LIN {X 5.578,Y -23.911,Z -42.731,A 0.015,B -0.000,C 180.000} C_DIS
LIN {X 5.597,Y -23.749,Z -43.353,A 0.015,B 0.000,C 180.000} C_DIS
LIN {X 5.625,Y -23.303,Z -43.816,A 0.015,B 0.000,C -180.000} C_DIS
LIN {X 5.610,Y -22.688,Z -44.000,A 0.015,B 0.000,C -180.000} C_DIS
LIN {X 1.585,Y -17.451,Z -44.244,A 0.015,B 0.000,C 180.000} C_DIS
LIN {X -4.825,Y -19.040,Z -44.488,A 0.015,B -0.000,C 180.000} C_DIS
LIN {X -5.938,Y -25.550,Z -44.732,A 0.015,B 0.000,C -180.000} C_DIS
LIN {X -0.420,Y -29.178,Z -44.976,A 0.015,B 0.000,C 180.000} C_DIS
LIN {X 5.116,Y -25.576,Z -45.220,A 0.015,B 0.000,C -180.000} C_DIS
LIN {X 4.034,Y -19.061,Z -45.464,A 0.015,B 0.000,C 180.000} C_DIS
LIN {X -2.368,Y -17.441,Z -45.708,A 0.015,B 0.000,C 180.000} C_DIS
LIN {X -6.418,Y -22.658,Z -45.952,A 0.015,B 0.000,C 180.000} C_DIS
LIN {X -3.261,Y -28.459,Z -46.196,A 0.015,B 0.000,C -180.000} C_DIS
LIN {X 3.319,Y -27.891,Z -46.440,A 0.015,B -0.000,C 180.000} C_DIS
LIN {X 5.435,Y -21.635,Z -46.685,A 0.015,B 0.000,C 180.000} C_DIS
LIN {X 0.551,Y -17.189,Z -46.929,A 0.015,B 0.000,C -180.000} C_DIS
LIN {X -5.479,Y -19.882,Z -47.173,A 0.015,B 0.000,C 180.000} C_DIS
LIN {X -5.428,Y -26.486,Z -47.417,A 0.015,B 0.000,C 180.000} C_DIS
LIN {X 0.643,Y -29.086,Z -47.661,A 0.015,B -0.000,C -180.000} C_DIS
LIN {X 5.458,Y -24.566,Z -47.905,A 0.015,B 0.000,C 180.000} C_DIS
LIN {X 3.245,Y -18.343,Z -48.149,A 0.015,B 0.000,C 180.000} C_DIS
LIN {X -3.342,Y -17.876,Z -48.393,A 0.015,B 0.000,C 180.000} C_DIS
LIN {X -6.410,Y -23.725,Z -48.637,A 0.015,B 0.000,C 180.000} C_DIS
LIN {X -2.281,Y -28.879,Z -48.881,A 0.015,B 0.000,C 180.000} C_DIS
LIN {X 4.096,Y -27.161,Z -49.125,A 0.015,B 0.000,C -180.000} C_DIS
LIN {X 5.078,Y -20.630,Z -49.369,A 0.015,B 0.000,C 180.000} C_DIS
LIN {X -0.513,Y -17.114,Z -49.613,A 0.015,B 0.000,C 180.000} C_DIS
LIN {X -5.974,Y -20.827,Z -49.857,A 0.015,B -0.000,C 180.000} C_DIS
LIN {X -4.761,Y -27.319,Z -50.101,A 0.015,B 0.000,C -180.000} C_DIS
LIN {X 1.673,Y -28.809,Z -50.345,A 0.015,B 0.000,C -180.000} C_DIS
LIN {X 5.616,Y -23.511,Z -50.589,A 0.015,B 0.000,C -180.000} C_DIS
LIN {X 2.342,Y -17.775,Z -50.833,A 0.015,B 0.000,C -180.000} C_DIS
LIN {X -4.225,Y -18.476,Z -51.077,A 0.015,B 0.000,C 180.000} C_DIS
LIN {X -6.214,Y -24.774,Z -51.321,A 0.015,B 0.000,C 180.000} C_DIS
LIN {X -1.241,Y -29.120,Z -51.565,A 0.015,B 0.000,C 180.000} C_DIS
LIN {X 4.733,Y -26.306,Z -51.810,A 0.015,B 0.000,C -180.000} C_DIS
LIN {X 4.549,Y -19.704,Z -52.054,A 0.015,B -0.000,C 180.000} C_DIS
LIN {X -1.573,Y -17.227,Z -52.298,A 0.015,B 0.000,C 180.000} C_DIS
LIN {X -6.296,Y -21.844,Z -52.542,A 0.015,B 0.000,C -180.000} C_DIS
LIN {X -3.958,Y -28.021,Z -52.786,A 0.015,B 0.000,C 180.000} C_DIS
LIN {X 2.638,Y -28.354,Z -53.030,A 0.015,B 0.000,C 180.000} C_DIS
LIN {X 5.586,Y -22.445,Z -53.274,A 0.015,B 0.000,C 180.000} C_DIS
LIN {X 1.354,Y -17.375,Z -53.518,A 0.015,B -0.000,C 180.000} C_DIS
LIN {X -4.987,Y -19.222,Z -53.762,A 0.015,B 0.000,C 180.000} C_DIS
LIN {X -5.836,Y -25.771,Z -54.006,A 0.015,B 0.000,C 180.000} C_DIS
LIN {X -0.176,Y -29.174,Z -54.250,A 0.015,B 0.000,C -180.000} C_DIS
LIN {X 5.210,Y -25.351,Z -54.494,A 0.015,B -0.000,C 180.000} C_DIS
LIN {X 3.865,Y -18.885,Z -54.738,A 0.015,B -0.000,C -180.000} C_DIS
LIN {X -2.597,Y -17.525,Z -54.982,A 0.015,B 0.000,C 180.000} C_DIS
LIN {X -6.433,Y -22.902,Z -55.226,A 0.015,B 0.000,C -180.000} C_DIS
LIN {X -3.044,Y -28.570,Z -55.470,A 0.015,B 0.000,C -180.000} C_DIS
LIN {X 3.508,Y -27.737,Z -55.714,A 0.015,B 0.000,C -180.000} C_DIS
LIN {X 5.369,Y -21.401,Z -55.958,A 0.015,B 0.000,C 180.000} C_DIS
LIN {X 0.310,Y -17.156,Z -56.202,A 0.015,B -0.000,C 180.000} C_DIS
LIN {X -5.607,Y -20.090,Z -56.446,A 0.015,B 0.000,C 180.000} C_DIS
LIN {X -5.289,Y -26.687,Z -56.690,A 0.015,B 0.000,C -180.000} C_DIS
LIN {X 0.882,Y -29.039,Z -56.935,A 0.015,B 0.000,C 180.000} C_DIS
LIN {X 5.510,Y -24.328,Z -57.179,A 0.015,B 0.000,C 180.000} C_DIS
LIN {X 3.048,Y -18.200,Z -57.423,A 0.015,B -0.000,C 180.000} C_DIS
LIN {X -3.553,Y -17.999,Z -57.667,A 0.015,B 0.000,C 180.000} C_DIS
LIN {X -6.382,Y -23.967,Z -57.911,A 0.015,B 0.000,C -180.000} C_DIS
LIN {X -2.047,Y -28.950,Z -58.155,A 0.015,B 0.000,C 180.000} C_DIS
LIN {X 4.255,Y -26.976,Z -58.399,A 0.015,B 0.000,C 180.000} C_DIS
LIN {X 4.972,Y -20.411,Z -58.643,A 0.015,B 0.000,C 180.000} C_DIS
LIN {X -0.756,Y -17.123,Z -58.887,A 0.015,B 0.000,C 180.000} C_DIS
LIN {X -6.064,Y -21.054,Z -59.131,A 0.015,B 0.000,C 180.000} C_DIS
LIN {X -4.589,Y -27.492,Z -59.375,A 0.015,B 0.000,C -180.000} C_DIS
LIN {X 1.900,Y -28.720,Z -59.619,A 0.015,B 0.000,C 180.000} C_DIS
LIN {X 5.626,Y -23.267,Z -59.863,A 0.015,B 0.000,C 180.000} C_DIS
LIN {X 2.123,Y -17.669,Z -60.107,A 0.015,B 0.000,C -180.000} C_DIS
LIN {X -4.410,Y -18.634,Z -60.351,A 0.015,B 0.000,C 180.000} C_DIS
LIN {X -6.143,Y -25.007,Z -60.595,A 0.015,B 0.000,C -180.000} C_DIS
LIN {X -0.999,Y -29.149,Z -60.839,A 0.015,B 0.000,C 180.000} C_DIS
LIN {X 4.857,Y -26.095,Z -61.083,A 0.015,B 0.000,C -180.000} C_DIS
LIN {X 4.406,Y -19.506,Z -61.327,A 0.015,B 0.000,C -180.000} C_DIS
LIN {X -1.812,Y -17.279,Z -61.571,A 0.015,B 0.000,C 180.000} C_DIS
LIN {X -6.344,Y -22.083,Z -61.815,A 0.015,B -0.000,C -180.000} C_DIS
LIN {X -3.758,Y -28.161,Z -62.060,A 0.015,B -0.000,C 180.000} C_DIS
LIN {X 2.846,Y -28.227,Z -62.304,A 0.015,B 0.000,C 180.000} C_DIS
LIN {X 5.553,Y -22.203,Z -62.548,A 0.015,B -0.000,C -180.000} C_DIS
LIN {X 1.119,Y -17.309,Z -62.792,A 0.015,B 0.000,C 180.000} C_DIS
LIN {X -5.142,Y -19.410,Z -63.036,A 0.015,B 0.000,C -180.000} C_DIS
LIN {X -5.726,Y -25.989,Z -63.280,A 0.015,B -0.000,C 180.000} C_DIS
LIN {X 0.067,Y -29.160,Z -63.524,A 0.015,B -0.000,C -180.000} C_DIS
LIN {X 5.294,Y -25.122,Z -63.768,A 0.015,B 0.000,C -180.000} C_DIS
LIN {X 3.690,Y -18.716,Z -64.012,A 0.015,B 0.000,C -180.000} C_DIS
LIN {X -2.823,Y -17.619,Z -64.256,A 0.015,B 0.000,C 180.000} C_DIS
LIN {X -6.438,Y -23.146,Z -64.500,A 0.015,B -0.000,C -180.000} C_DIS
CIRC {X -0.832,Y -28.751,Z -64.500,A 0.015,B 0.000,C -180.000},{X 4.774,Y -23.145,Z -64.500,A 0.015,B 0.000,C 180.000} C_DIS
LIN {X 4.774,Y -20.361,Z -64.500,A 0.015,B 0.000,C -180.000} C_DIS
CIRC {X 3.668,Y -18.804,Z -64.500,A 0.015,B 0.000,C -180.000},{X 1.834,Y -19.336,Z -64.500,A 0.015,B -0.000,C -180.000} C_DIS
LIN {X -0.747,Y -22.588,Z -64.500,A 0.015,B -0.000,C 180.000} C_DIS
CIRC {X -0.977,Y -24.658,Z -64.500,A 0.015,B 0.000,C 180.000},{X 0.787,Y -25.765,Z -64.500,A 0.015,B -0.000,C 180.000} C_DIS
LIN {X 2.660,Y -25.765,Z -64.500,A 0.015,B 0.000,C -180.000} C_DIS
CIRC {X 4.155,Y -25.146,Z -64.500,A 0.015,B -0.000,C 180.000},{X 4.774,Y -23.651,Z -64.500,A 0.015,B 0.000,C -180.000} C_DIS
LIN {X 4.774,Y -23.145,Z -64.500,A 0.015,B -0.000,C 180.000} C_DIS
LIN {X 3.563,Y -23.413,Z -64.500,A 0.015,B 0.000,C 180.000} C_DIS
LIN {X 4.057,Y -24.474,Z -64.500,A 0.015,B 0.000,C 180.000} C_DIS
LIN {X 4.252,Y -24.715,Z -64.500,A 0.015,B 0.000,C -180.000} C_DIS
LIN {X 8.679,Y -28.027,Z -64.500,A 0.015,B -0.000,C 180.000} C_DIS
LIN {X 9.366,Y -28.668,Z -64.500,A 0.015,B 0.000,C -180.000} C_DIS
LIN {X 9.675,Y -28.604,Z -64.500,A 0.015,B 0.000,C -180.000} C_DIS
LIN {X 10.021,Y -27.803,Z -64.500,A 0.015,B 0.000,C -180.000} C_DIS
LIN {X 10.218,Y -26.938,Z -64.500,A 0.015,B -0.000,C 180.000} C_DIS
LIN {X 10.275,Y -25.867,Z -64.500,A 0.015,B 0.000,C -180.000} C_DIS
LIN {X 10.274,Y 7.389,Z -64.500,A 0.015,B -0.000,C 180.000} C_DIS
LIN {X 6.193,Y -2.899,Z -64.500,A 0.015,B 0.000,C -180.000} C_DIS
LIN {X 5.976,Y -3.347,Z -64.500,A 0.015,B 0.000,C 180.000} C_DIS
LIN {X 1.986,Y -10.239,Z -64.500,A 0.015,B -0.000,C 180.000} C_DIS
LIN {X 1.708,Y -10.647,Z -64.500,A 0.015,B -0.000,C 180.000} C_DIS
LIN {X -5.904,Y -20.237,Z -64.500,A 0.015,B 0.000,C -180.000} C_DIS
LIN {X -6.318,Y -20.673,Z -64.500,A 0.015,B -0.000,C -180.000} C_DIS
LIN {X -7.322,Y -21.557,Z -64.500,A 0.015,B -0.000,C 180.000} C_DIS
LIN {X -7.657,Y -21.816,Z -64.500,A 0.015,B -0.000,C 180.000} C_DIS
LIN {X -17.247,Y -28.331,Z -64.500,A 0.015,B 0.000,C 180.000} C_DIS
LIN {X -17.736,Y -28.607,Z -64.500,A 0.015,B 0.000,C -180.000} C_DIS
LIN {X -19.187,Y -29.273,Z -64.500,A 0.015,B 0.000,C -180.000} C_DIS
LIN {X -19.614,Y -29.435,Z -64.500,A 0.015,B -0.000,C 180.000} C_DIS
LIN {X -25.630,Y -31.266,Z -64.500,A 0.015,B 0.000,C 180.000} C_DIS
LIN {X 5.412,Y -31.266,Z -64.500,A 0.015,B 0.000,C 180.000} C_DIS
LIN {X 6.622,Y -31.073,Z -64.500,A 0.015,B 0.000,C 180.000} C_DIS
$VEL.CP = 1.00000
LIN {X 6.622,Y -31.073,Z 11.769,A 0.015,B 0.000,C -180.000} C_DIS
$VEL.CP = 1.00000
LIN {X -399.068,Y -22.363,Z 11.769,A 0.015,B 0.000,C -180.000} C_DIS
$VEL.CP = 0.10000
LIN {X -399.086,Y -22.525,Z 11.147,A 0.015,B 0.000,C -180.000} C_DIS
LIN {X -399.115,Y -22.971,Z 10.684,A 0.015,B -0.000,C 180.000} C_DIS
LIN {X -399.099,Y -23.586,Z 10.500,A 0.015,B -0.000,C -180.000} C_DIS
LIN {X -395.075,Y -28.823,Z 10.256,A 0.015,B 0.000,C 180.000} C_DIS
LIN {X -388.665,Y -27.234,Z 10.012,A 0.015,B -0.000,C 180.000} C_DIS
LIN {X -387.551,Y -20.725,Z 9.768,A 0.015,B 0.000,C 180.000} C_DIS
LIN {X -393.069,Y -17.096,Z 9.524,A 0.015,B 0.000,C 180.000} C_DIS
LIN {X -398.605,Y -20.698,Z 9.280,A 0.015,B -0.000,C 180.000} C_DIS
LIN {X -397.524,Y -27.213,Z 9.036,A 0.015,B -0.000,C -180.000} C_DIS
LIN {X -391.121,Y -28.833,Z 8.792,A 0.015,B 0.000,C -180.000} C_DIS
LIN {X -387.071,Y -23.616,Z 8.548,A 0.015,B -0.000,C -180.000} C_DIS
LIN {X -390.228,Y -17.815,Z 8.304,A 0.015,B 0.000,C -180.000} C_DIS
LIN {X -396.808,Y -18.383,Z 8.060,A 0.015,B 0.000,C 180.000} C_DIS
LIN {X -398.925,Y -24.639,Z 7.815,A 0.015,B 0.000,C -180.000} C_DIS
LIN {X -394.041,Y -29.085,Z 7.571,A 0.015,B -0.000,C -180.000} C_DIS
LIN {X -388.011,Y -26.392,Z 7.327,A 0.015,B -0.000,C -180.000} C_DIS
LIN {X -388.061,Y -19.788,Z 7.083,A 0.015,B -0.000,C -180.000} C_DIS
LIN {X -394.132,Y -17.188,Z 6.839,A 0.015,B 0.000,C 180.000} C_DIS
LIN {X -398.947,Y -21.708,Z 6.595,A 0.015,B 0.000,C 180.000} C_DIS
LIN {X -396.735,Y -27.931,Z 6.351,A 0.015,B 0.000,C 180.000} C_DIS
LIN {X -390.147,Y -28.398,Z 6.107,A 0.015,B -0.000,C 180.000} C_DIS
LIN {X -387.080,Y -22.549,Z 5.863,A 0.015,B 0.000,C 180.000} C_DIS
LIN {X -391.209,Y -17.395,Z 5.619,A 0.015,B -0.000,C -180.000} C_DIS
LIN {X -397.586,Y -19.113,Z 5.375,A 0.015,B -0.000,C -180.000} C_DIS
LIN {X -398.567,Y -25.644,Z 5.131,A 0.015,B -0.000,C -180.000} C_DIS
LIN {X -392.977,Y -29.160,Z 4.887,A 0.015,B 0.000,C -180.000} C_DIS
LIN {X -387.515,Y -25.447,Z 4.643,A 0.015,B 0.000,C 180.000} C_DIS
LIN {X -388.728,Y -18.955,Z 4.399,A 0.015,B 0.000,C -180.000} C_DIS
LIN {X -395.162,Y -17.465,Z 4.155,A 0.015,B -0.000,C -180.000} C_DIS
LIN {X -399.106,Y -22.763,Z 3.911,A 0.015,B -0.000,C 180.000} C_DIS
LIN {X -395.832,Y -28.499,Z 3.667,A 0.015,B 0.000,C 180.000} C_DIS
LIN {X -389.265,Y -27.798,Z 3.423,A 0.015,B 0.000,C -180.000} C_DIS
LIN {X -387.275,Y -21.501,Z 3.179,A 0.015,B -0.000,C 180.000} C_DIS
LIN {X -392.248,Y -17.154,Z 2.935,A 0.015,B -0.000,C -180.000} C_DIS
LIN {X -398.223,Y -19.968,Z 2.690,A 0.015,B -0.000,C -180.000} C_DIS
LIN {X -398.039,Y -26.570,Z 2.446,A 0.015,B 0.000,C -180.000} C_DIS
LIN {X -391.916,Y -29.047,Z 2.202,A 0.015,B 0.000,C -180.000} C_DIS
LIN {X -387.194,Y -24.430,Z 1.958,A 0.015,B 0.000,C -180.000} C_DIS
LIN {X -389.531,Y -18.253,Z 1.714,A 0.015,B 0.000,C -180.000} C_DIS
LIN {X -396.127,Y -17.920,Z 1.470,A 0.015,B 0.000,C -180.000} C_DIS
LIN {X -399.076,Y -23.829,Z 1.226,A 0.015,B -0.000,C 180.000} C_DIS
LIN {X -394.843,Y -28.899,Z 0.982,A 0.015,B 0.000,C 180.000} C_DIS
LIN {X -388.502,Y -27.052,Z 0.738,A 0.015,B 0.000,C -180.000} C_DIS
LIN {X -387.653,Y -20.503,Z 0.494,A 0.015,B -0.000,C 180.000} C_DIS
LIN {X -393.313,Y -17.100,Z 0.250,A 0.015,B 0.000,C -180.000} C_DIS
LIN {X -398.699,Y -20.923,Z 0.006,A 0.015,B 0.000,C 180.000} C_DIS
LIN {X -397.355,Y -27.389,Z -0.238,A 0.015,B -0.000,C -180.000} C_DIS
LIN {X -390.892,Y -28.749,Z -0.482,A 0.015,B 0.000,C -180.000} C_DIS
LIN {X -387.057,Y -23.372,Z -0.726,A 0.015,B 0.000,C 180.000} C_DIS
LIN {X -390.445,Y -17.704,Z -0.970,A 0.015,B -0.000,C 180.000} C_DIS
LIN {X -396.997,Y -18.537,Z -1.214,A 0.015,B 0.000,C 180.000} C_DIS
LIN {X -398.859,Y -24.874,Z -1.458,A 0.015,B 0.000,C -180.000} C_DIS
LIN {X -393.799,Y -29.119,Z -1.702,A 0.015,B -0.000,C -180.000} C_DIS
LIN {X -387.883,Y -26.184,Z -1.946,A 0.015,B 0.000,C -180.000} C_DIS
LIN {X -388.200,Y -19.587,Z -2.190,A 0.015,B 0.000,C 180.000} C_DIS
LIN {X -394.372,Y -17.235,Z -2.435,A 0.015,B 0.000,C 180.000} C_DIS
LIN {X -399.000,Y -21.946,Z -2.679,A 0.015,B -0.000,C 180.000} C_DIS
LIN {X -396.538,Y -28.075,Z -2.923,A 0.015,B 0.000,C 180.000} C_DIS
LIN {X -389.936,Y -28.275,Z -3.167,A 0.015,B 0.000,C -180.000} C_DIS
LIN {X -387.108,Y -22.307,Z -3.411,A 0.015,B -0.000,C 180.000} C_DIS
LIN {X -391.442,Y -17.324,Z -3.655,A 0.015,B 0.000,C -180.000} C_DIS
LIN {X -397.745,Y -19.298,Z -3.899,A 0.015,B -0.000,C -180.000} C_DIS
LIN {X -398.461,Y -25.863,Z -4.143,A 0.015,B -0.000,C 180.000} C_DIS
LIN {X -392.733,Y -29.151,Z -4.387,A 0.015,B 0.000,C 180.000} C_DIS
LIN {X -387.426,Y -25.220,Z -4.631,A 0.015,B 0.000,C 180.000} C_DIS
LIN {X -388.900,Y -18.783,Z -4.875,A 0.015,B 0.000,C -180.000} C_DIS
LIN {X -395.389,Y -17.554,Z -5.119,A 0.015,B -0.000,C -180.000} C_DIS
LIN {X -399.115,Y -23.007,Z -5.363,A 0.015,B 0.000,C 180.000} C_DIS
LIN {X -395.613,Y -28.606,Z -5.607,A 0.015,B -0.000,C -180.000} C_DIS
LIN {X -389.079,Y -27.640,Z -5.851,A 0.015,B -0.000,C 180.000} C_DIS
LIN {X -387.346,Y -21.267,Z -6.095,A 0.015,B -0.000,C -180.000} C_DIS
LIN {X -392.490,Y -17.125,Z -6.339,A 0.015,B -0.000,C -180.000} C_DIS
LIN {X -398.346,Y -20.179,Z -6.583,A 0.015,B 0.000,C 180.000} C_DIS
LIN {X -397.895,Y -26.768,Z -6.827,A 0.015,B -0.000,C -180.000} C_DIS
LIN {X -391.678,Y -28.995,Z -7.071,A 0.015,B -0.000,C 180.000} C_DIS
LIN {X -387.146,Y -24.191,Z -7.315,A 0.015,B 0.000,C -180.000} C_DIS
LIN {X -389.731,Y -18.114,Z -7.560,A 0.015,B -0.000,C -180.000} C_DIS
LIN {X -396.335,Y -18.047,Z -7.804,A 0.015,B -0.000,C 180.000} C_DIS
LIN {X -399.043,Y -24.071,Z -8.048,A 0.015,B -0.000,C 180.000} C_DIS
LIN {X -394.608,Y -28.965,Z -8.292,A 0.015,B -0.000,C -180.000} C_DIS
LIN {X -388.347,Y -26.864,Z -8.536,A 0.015,B -0.000,C 180.000} C_DIS
LIN {X -387.764,Y -20.286,Z -8.780,A 0.015,B -0.000,C -180.000} C_DIS
LIN {X -393.557,Y -17.115,Z -9.024,A 0.015,B -0.000,C 180.000} C_DIS
LIN {X -398.784,Y -21.152,Z -9.268,A 0.015,B -0.000,C 180.000} C_DIS
LIN {X -397.179,Y -27.558,Z -9.512,A 0.015,B 0.000,C -180.000} C_DIS
LIN {X -390.667,Y -28.655,Z -9.756,A 0.015,B 0.000,C -180.000} C_DIS
LIN {X -387.052,Y -23.128,Z -10.000,A 0.015,B -0.000,C -180.000} C_DIS
CIRC {X -388.694,Y -19.164,Z -10.000,A 0.015,B 0.000,C -180.000},{X -392.658,Y -17.522,Z -10.000,A 0.015,B 0.000,C 180.000} C_DIS
CIRC {X -396.623,Y -19.164,Z -10.000,A 0.015,B 0.000,C 180.000},{X -398.265,Y -23.129,Z -10.000,A 0.015,B 0.000,C 180.000} C_DIS
LIN {X -398.265,Y -23.640,Z -10.000,A 0.015,B 0.000,C 180.000} C_DIS
CIRC {X -397.646,Y -25.134,Z -10.000,A 0.015,B -0.000,C 180.000},{X -396.151,Y -25.754,Z -10.000,A 0.015,B -0.000,C 180.000} C_DIS
LIN {X -394.248,Y -25.754,Z -10.000,A 0.015,B -0.000,C 180.000} C_DIS
CIRC {X -392.485,Y -24.645,Z -10.000,A 0.015,B 0.000,C 180.000},{X -392.720,Y -22.577,Z -10.000,A 0.015,B 0.000,C -180.000} C_DIS
LIN {X -395.322,Y -19.323,Z -10.000,A 0.015,B -0.000,C -180.000} C_DIS
CIRC {X -397.159,Y -18.795,Z -10.000,A 0.015,B -0.000,C 180.000},{X -398.265,Y -20.354,Z -10.000,A 0.015,B -0.000,C -180.000} C_DIS
LIN {X -398.265,Y -23.129,Z -10.000,A 0.015,B 0.000,C 180.000} C_DIS
LIN {X -398.413,Y -23.653,Z -10.000,A 0.015,B 0.000,C 180.000} C_DIS
LIN {X -401.465,Y -28.615,Z -10.000,A 0.015,B -0.000,C 180.000} C_DIS
CIRC {X -402.315,Y -29.091,Z -10.000,A 0.015,B -0.000,C 180.000},{X -403.166,Y -28.618,Z -10.000,A 0.015,B 0.000,C -180.000} C_DIS
LIN {X -403.274,Y -28.444,Z -10.000,A 0.015,B -0.000,C 180.000} C_DIS
LIN {X -403.584,Y -27.623,Z -10.000,A 0.015,B 0.000,C 180.000} C_DIS
LIN {X -403.777,Y -26.414,Z -10.000,A 0.015,B -0.000,C 180.000} C_DIS
LIN {X -403.778,Y 7.612,Z -10.000,A 0.015,B -0.000,C 180.000} C_DIS
LIN {X -399.888,Y -2.503,Z -10.000,A 0.015,B 0.000,C 180.000} C_DIS
LIN {X -399.667,Y -2.969,Z -10.000,A 0.015,B 0.000,C -180.000} C_DIS
LIN {X -395.598,Y -10.084,Z -10.000,A 0.015,B 0.000,C 180.000} C_DIS
LIN {X -395.303,Y -10.517,Z -10.000,A 0.015,B -0.000,C -180.000} C_DIS
LIN {X -387.527,Y -20.246,Z -10.000,A 0.015,B 0.000,C 180.000} C_DIS
LIN {X -387.304,Y -20.498,Z -10.000,A 0.015,B -0.000,C 180.000} C_DIS
LIN {X -386.606,Y -21.212,Z -10.000,A 0.015,B -0.000,C 180.000} C_DIS
LIN {X -386.065,Y -21.661,Z -10.000,A 0.015,B 0.000,C 180.000} C_DIS
LIN {X -376.242,Y -28.219,Z -10.000,A 0.015,B 0.000,C 180.000} C_DIS
LIN {X -376.074,Y -28.324,Z -10.000,A 0.015,B -0.000,C 180.000} C_DIS
LIN {X -374.907,Y -29.008,Z -10.000,A 0.015,B 0.000,C 180.000} C_DIS
LIN {X -374.141,Y -29.338,Z -10.000,A 0.015,B 0.000,C 180.000} C_DIS
LIN {X -367.506,Y -31.266,Z -10.000,A 0.015,B 0.000,C 180.000} C_DIS
LIN {X -398.962,Y -31.266,Z -10.000,A 0.015,B -0.000,C -180.000} C_DIS
LIN {X -399.885,Y -31.140,Z -10.000,A 0.015,B -0.000,C -180.000} C_DIS
LIN {X -400.741,Y -30.861,Z -10.000,A 0.015,B 0.000,C 180.000} C_DIS
LIN {X -401.186,Y -30.616,Z -10.000,A 0.015,B 0.000,C -180.000} C_DIS
LIN {X -401.261,Y -29.553,Z -10.000,A 0.015,B 0.000,C 180.000} C_DIS
LIN {X -398.545,Y -27.507,Z -10.000,A 0.015,B 0.000,C 180.000} C_DIS
LIN {X -393.929,Y -23.873,Z -10.000,A 0.015,B 0.000,C -180.000} C_DIS
LIN {X -392.175,Y -23.277,Z -10.000,A 0.015,B 0.000,C -180.000} C_DIS
LIN {X -391.930,Y -22.788,Z -10.000,A 0.015,B 0.000,C 180.000} C_DIS
LIN {X -397.126,Y -18.717,Z -10.244,A 0.015,B -0.000,C 180.000} C_DIS
LIN {X -402.940,Y -21.842,Z -10.488,A 0.015,B 0.000,C -180.000} C_DIS
LIN {X -402.411,Y -28.421,Z -10.732,A 0.015,B 0.000,C -180.000} C_DIS
LIN {X -396.173,Y -30.578,Z -10.976,A 0.015,B -0.000,C 180.000} C_DIS
LIN {X -391.694,Y -25.729,Z -11.220,A 0.015,B -0.000,C 180.000} C_DIS
LIN {X -394.337,Y -19.680,Z -11.463,A 0.015,B 0.000,C -180.000} C_DIS
LIN {X -400.938,Y -19.674,Z -11.707,A 0.015,B -0.000,C -180.000} C_DIS
LIN {X -403.593,Y -25.718,Z -11.951,A 0.015,B -0.000,C -180.000} C_DIS
LIN {X -399.123,Y -30.575,Z -12.195,A 0.015,B 0.000,C -180.000} C_DIS
LIN {X -392.881,Y -28.430,Z -12.439,A 0.015,B -0.000,C 180.000} C_DIS
LIN {X -392.339,Y -21.852,Z -12.683,A 0.015,B -0.000,C 180.000} C_DIS
LIN {X -398.147,Y -18.716,Z -12.927,A 0.015,B 0.000,C -180.000} C_DIS
LIN {X -403.351,Y -22.777,Z -13.171,A 0.015,B -0.000,C -180.000} C_DIS
LIN {X -401.720,Y -29.173,Z -13.415,A 0.015,B -0.000,C -180.000} C_DIS
LIN {X -395.207,Y -30.246,Z -13.659,A 0.015,B 0.000,C -180.000} C_DIS
LIN {X -391.610,Y -24.711,Z -13.902,A 0.015,B 0.000,C -180.000} C_DIS
LIN {X -395.236,Y -19.195,Z -14.146,A 0.015,B 0.000,C 180.000} C_DIS
LIN {X -401.743,Y -20.302,Z -14.390,A 0.015,B 0.000,C -180.000} C_DIS
LIN {X -403.341,Y -26.707,Z -14.634,A 0.015,B 0.000,C 180.000} C_DIS
LIN {X -398.116,Y -30.741,Z -14.878,A 0.015,B 0.000,C -180.000} C_DIS
LIN {X -392.324,Y -27.574,Z -15.122,A 0.015,B 0.000,C -180.000} C_DIS
LIN {X -392.900,Y -20.999,Z -15.366,A 0.015,B 0.000,C 180.000} C_DIS
LIN {X -399.154,Y -18.887,Z -15.610,A 0.015,B 0.000,C -180.000} C_DIS
LIN {X -403.598,Y -23.767,Z -15.854,A 0.015,B -0.000,C 180.000} C_DIS
LIN {X -400.912,Y -29.797,Z -16.098,A 0.015,B 0.000,C 180.000} C_DIS
LIN {X -394.311,Y -29.756,Z -16.341,A 0.015,B 0.000,C -180.000} C_DIS
LIN {X -391.699,Y -23.694,Z -16.585,A 0.015,B -0.000,C 180.000} C_DIS
LIN {X -396.203,Y -18.869,Z -16.829,A 0.015,B 0.000,C 180.000} C_DIS
LIN {X -402.430,Y -21.057,Z -17.073,A 0.015,B 0.000,C 180.000} C_DIS
LIN {X -402.925,Y -27.640,Z -17.317,A 0.015,B 0.000,C -180.000} C_DIS
LIN {X -397.095,Y -30.735,Z -17.561,A 0.015,B -0.000,C 180.000} C_DIS
LIN {X -391.920,Y -26.636,Z -17.805,A 0.015,B -0.000,C 180.000} C_DIS
LIN {X -393.597,Y -20.252,Z -18.049,A 0.015,B 0.000,C -180.000} C_DIS
LIN {X -400.117,Y -19.225,Z -18.293,A 0.015,B 0.000,C -180.000} C_DIS
LIN {X -403.675,Y -24.786,Z -18.537,A 0.015,B 0.000,C -180.000} C_DIS
LIN {X -400.010,Y -30.276,Z -18.780,A 0.015,B 0.000,C 180.000} C_DIS
LIN {X -393.510,Y -29.122,Z -19.024,A 0.015,B -0.000,C 180.000} C_DIS
LIN {X -391.958,Y -22.706,Z -19.268,A 0.015,B 0.000,C -180.000} C_DIS
LIN {X -397.212,Y -18.710,Z -19.512,A 0.015,B 0.000,C 180.000} C_DIS
LIN {X -402.981,Y -21.918,Z -19.756,A 0.015,B 0.000,C -180.000} C_DIS
LIN {X -402.358,Y -28.489,Z -20.000,A 0.015,B -0.000,C -180.000} C_DIS
CIRC {X -398.602,Y -30.564,Z -20.000,A 0.015,B -0.000,C -180.000},{X -394.479,Y -29.375,Z -20.000,A 0.015,B -0.000,C -180.000} C_DIS
CIRC {X -392.404,Y -25.619,Z -20.000,A 0.015,B 0.000,C 180.000},{X -393.593,Y -21.496,Z -20.000,A 0.015,B 0.000,C -180.000} C_DIS
LIN {X -395.325,Y -19.325,Z -20.000,A 0.015,B 0.000,C -180.000} C_DIS
CIRC {X -397.162,Y -18.796,Z -20.000,A 0.015,B 0.000,C -180.000},{X -398.268,Y -20.354,Z -20.000,A 0.015,B 0.000,C -180.000} C_DIS
LIN {X -398.267,Y -23.642,Z -20.000,A 0.015,B 0.000,C -180.000} C_DIS
CIRC {X -397.648,Y -25.137,Z -20.000,A 0.015,B 0.000,C -180.000},{X -396.154,Y -25.756,Z -20.000,A 0.015,B 0.000,C -180.000} C_DIS
LIN {X -394.258,Y -25.756,Z -20.000,A 0.015,B 0.000,C -180.000} C_DIS
CIRC {X -392.495,Y -24.648,Z -20.000,A 0.015,B 0.000,C -180.000},{X -392.729,Y -22.579,Z -20.000,A 0.015,B -0.000,C 180.000} C_DIS
LIN {X -393.593,Y -21.496,Z -20.000,A 0.015,B 0.000,C -180.000} C_DIS
CIRC {X -394.365,Y -21.120,Z -20.000,A 0.015,B -0.000,C -180.000},{X -395.144,Y -21.481,Z -20.000,A 0.015,B 0.000,C 180.000} C_DIS
LIN {X -401.471,Y -29.102,Z -20.000,A 0.015,B -0.000,C 180.000} C_DIS
LIN {X -401.186,Y -30.616,Z -20.000,A 0.015,B 0.000,C 180.000} C_DIS
LIN {X -400.741,Y -30.861,Z -20.000,A 0.015,B 0.000,C 180.000} C_DIS
LIN {X -399.885,Y -31.140,Z -20.000,A 0.015,B 0.000,C -180.000} C_DIS
LIN {X -398.962,Y -31.266,Z -20.000,A 0.015,B -0.000,C 180.000} C_DIS
LIN {X -367.621,Y -31.266,Z -20.000,A 0.015,B 0.000,C 180.000} C_DIS
LIN {X -373.860,Y -29.446,Z -20.000,A 0.015,B 0.000,C -180.000} C_DIS
LIN {X -374.354,Y -29.260,Z -20.000,A 0.015,B 0.000,C -180.000} C_DIS
LIN {X -375.363,Y -28.784,Z -20.000,A 0.015,B 0.000,C 180.000} C_DIS
LIN {X -375.806,Y -28.534,Z -20.000,A 0.015,B 0.000,C 180.000} C_DIS
LIN {X -386.074,Y -21.655,Z -20.000,A 0.015,B 0.000,C -180.000} C_DIS
LIN {X -386.585,Y -21.234,Z -20.000,A 0.015,B 0.000,C -180.000} C_DIS
LIN {X -387.294,Y -20.524,Z -20.000,A 0.015,B -0.000,C 180.000} C_DIS
LIN {X -387.544,Y -20.243,Z -20.000,A 0.015,B -0.000,C 180.000} C_DIS
LIN {X -395.306,Y -10.515,Z -20.000,A 0.015,B 0.000,C 180.000} C_DIS
LIN {X -395.598,Y -10.084,Z -20.000,A 0.015,B -0.000,C 180.000} C_DIS
LIN {X -399.667,Y -2.969,Z -20.000,A 0.015,B 0.000,C 180.000} C_DIS
LIN {X -399.884,Y -2.512,Z -20.000,A 0.015,B -0.000,C -180.000} C_DIS
LIN {X -403.778,Y 7.527,Z -20.000,A 0.015,B -0.000,C 180.000} C_DIS
LIN {X -403.777,Y -26.414,Z -20.000,A 0.015,B 0.000,C 180.000} C_DIS
LIN {X -403.584,Y -27.623,Z -20.000,A 0.015,B 0.000,C 180.000} C_DIS
LIN {X -403.274,Y -28.444,Z -20.000,A 0.015,B -0.000,C -180.000} C_DIS
$VEL.CP = 1.00000
LIN {X -403.274,Y -28.444,Z 11.000,A 0.015,B 0.000,C 180.000} C_DIS
$VEL.CP = 1.00000
LIN {X -399.074,Y -22.371,Z 11.000,A 0.015,B -0.000,C -180.000} C_DIS
$VEL.CP = 0.10000
LIN {X -399.074,Y -22.371,Z -8.231,A 0.015,B 0.000,C -180.000} C_DIS
LIN {X -399.092,Y -22.533,Z -8.853,A 0.015,B -0.000,C -180.000} C_DIS
LIN {X -399.121,Y -22.979,Z -9.316,A 0.015,B 0.000,C -180.000} C_DIS
LIN {X -399.105,Y -23.594,Z -9.500,A 0.015,B -0.000,C 180.000} C_DIS
LIN {X -395.081,Y -28.831,Z -9.744,A 0.015,B -0.000,C -180.000} C_DIS
LIN {X -388.671,Y -27.242,Z -9.988,A 0.015,B -0.000,C 180.000} C_DIS
LIN {X -387.557,Y -20.733,Z -10.232,A 0.015,B -0.000,C 180.000} C_DIS
LIN {X -393.075,Y -17.104,Z -10.476,A 0.015,B 0.000,C -180.000} C_DIS
LIN {X -398.611,Y -20.706,Z -10.720,A 0.015,B 0.000,C 180.000} C_DIS
LIN {X -397.530,Y -27.221,Z -10.964,A 0.015,B -0.000,C 180.000} C_DIS
LIN {X -391.127,Y -28.841,Z -11.208,A 0.015,B -0.000,C -180.000} C_DIS
LIN {X -387.077,Y -23.624,Z -11.452,A 0.015,B 0.000,C 180.000} C_DIS
LIN {X -390.234,Y -17.823,Z -11.696,A 0.015,B 0.000,C -180.000} C_DIS
LIN {X -396.814,Y -18.391,Z -11.940,A 0.015,B -0.000,C 180.000} C_DIS
LIN {X -398.931,Y -24.647,Z -12.185,A 0.015,B -0.000,C 180.000} C_DIS
LIN {X -394.047,Y -29.093,Z -12.429,A 0.015,B 0.000,C -180.000} C_DIS
LIN {X -388.016,Y -26.400,Z -12.673,A 0.015,B 0.000,C 180.000} C_DIS
LIN {X -388.067,Y -19.796,Z -12.917,A 0.015,B 0.000,C 180.000} C_DIS
LIN {X -394.138,Y -17.196,Z -13.161,A 0.015,B 0.000,C 180.000} C_DIS
LIN {X -398.953,Y -21.716,Z -13.405,A 0.015,B 0.000,C -180.000} C_DIS
LIN {X -396.741,Y -27.939,Z -13.649,A 0.015,B 0.000,C 180.000} C_DIS
LIN {X -390.153,Y -28.406,Z -13.893,A 0.015,B 0.000,C 180.000} C_DIS
LIN {X -387.086,Y -22.557,Z -14.137,A 0.015,B 0.000,C 180.000} C_DIS
LIN {X -391.215,Y -17.403,Z -14.381,A 0.015,B 0.000,C 180.000} C_DIS
LIN {X -397.592,Y -19.121,Z -14.625,A 0.015,B 0.000,C -180.000} C_DIS
LIN {X -398.573,Y -25.652,Z -14.869,A 0.015,B 0.000,C 180.000} C_DIS
LIN {X -392.983,Y -29.168,Z -15.113,A 0.015,B 0.000,C 180.000} C_DIS
LIN {X -387.521,Y -25.455,Z -15.357,A 0.015,B 0.000,C 180.000} C_DIS
LIN {X -388.734,Y -18.963,Z -15.601,A 0.015,B 0.000,C 180.000} C_DIS
LIN {X -395.168,Y -17.473,Z -15.845,A 0.015,B -0.000,C -180.000} C_DIS
LIN {X -399.112,Y -22.771,Z -16.089,A 0.015,B 0.000,C 180.000} C_DIS
LIN {X -395.838,Y -28.507,Z -16.333,A 0.015,B 0.000,C 180.000} C_DIS
LIN {X -389.271,Y -27.806,Z -16.577,A 0.015,B 0.000,C -180.000} C_DIS
LIN {X -387.281,Y -21.508,Z -16.821,A 0.015,B 0.000,C 180.000} C_DIS
LIN {X -392.254,Y -17.162,Z -17.065,A 0.015,B 0.000,C -180.000} C_DIS
LIN {X -398.229,Y -19.976,Z -17.310,A 0.015,B 0.000,C 180.000} C_DIS
LIN {X -398.044,Y -26.578,Z -17.554,A 0.015,B -0.000,C 180.000} C_DIS
LIN {X -391.922,Y -29.055,Z -17.798,A 0.015,B 0.000,C -180.000} C_DIS
LIN {X -387.200,Y -24.438,Z -18.042,A 0.015,B -0.000,C 180.000} C_DIS
LIN {X -389.537,Y -18.261,Z -18.286,A 0.015,B -0.000,C -180.000} C_DIS
LIN {X -396.133,Y -17.928,Z -18.530,A 0.015,B 0.000,C 180.000} C_DIS
LIN {X -399.082,Y -23.837,Z -18.774,A 0.015,B -0.000,C -180.000} C_DIS
LIN {X -394.849,Y -28.907,Z -19.018,A 0.015,B 0.000,C 180.000} C_DIS
LIN {X -388.508,Y -27.060,Z -19.262,A 0.015,B 0.000,C 180.000} C_DIS
LIN {X -387.659,Y -20.511,Z -19.506,A 0.015,B 0.000,C -180.000} C_DIS
LIN {X -393.319,Y -17.108,Z -19.750,A 0.015,B 0.000,C -180.000} C_DIS
LIN {X -398.705,Y -20.931,Z -19.994,A 0.015,B 0.000,C -180.000} C_DIS
LIN {X -397.361,Y -27.397,Z -20.238,A 0.015,B -0.000,C -180.000} C_DIS
LIN {X -390.898,Y -28.757,Z -20.482,A 0.015,B -0.000,C -180.000} C_DIS
LIN {X -387.063,Y -23.380,Z -20.726,A 0.015,B 0.000,C -180.000} C_DIS
LIN {X -390.451,Y -17.712,Z -20.970,A 0.015,B -0.000,C -180.000} C_DIS
LIN {X -397.003,Y -18.545,Z -21.214,A 0.015,B -0.000,C 180.000} C_DIS
LIN {X -398.865,Y -24.882,Z -21.458,A 0.015,B 0.000,C -180.000} C_DIS
LIN {X -393.805,Y -29.126,Z -21.702,A 0.015,B 0.000,C -180.000} C_DIS
LIN {X -387.889,Y -26.192,Z -21.946,A 0.015,B 0.000,C -180.000} C_DIS
LIN {X -388.206,Y -19.595,Z -22.190,A 0.015,B -0.000,C 180.000} C_DIS
LIN {X -394.377,Y -17.243,Z -22.435,A 0.015,B 0.000,C -180.000} C_DIS
LIN {X -399.006,Y -21.954,Z -22.679,A 0.015,B 0.000,C 180.000} C_DIS
LIN {X -396.544,Y -28.083,Z -22.923,A 0.015,B -0.000,C -180.000} C_DIS
LIN {X -389.942,Y -28.283,Z -23.167,A 0.015,B 0.000,C 180.000} C_DIS
LIN {X -387.114,Y -22.315,Z -23.411,A 0.015,B 0.000,C -180.000} C_DIS
LIN {X -391.448,Y -17.332,Z -23.655,A 0.015,B -0.000,C 180.000} C_DIS
LIN {X -397.750,Y -19.306,Z -23.899,A 0.015,B 0.000,C 180.000} C_DIS
LIN {X -398.467,Y -25.871,Z -24.143,A 0.015,B -0.000,C 180.000} C_DIS
LIN {X -392.739,Y -29.159,Z -24.387,A 0.015,B 0.000,C 180.000} C_DIS
LIN {X -387.432,Y -25.228,Z -24.631,A 0.015,B 0.000,C -180.000} C_DIS
LIN {X -388.906,Y -18.790,Z -24.875,A 0.015,B 0.000,C 180.000} C_DIS
LIN {X -395.395,Y -17.562,Z -25.119,A 0.015,B 0.000,C 180.000} C_DIS
LIN {X -399.121,Y -23.015,Z -25.363,A 0.015,B -0.000,C -180.000} C_DIS
LIN {X -395.619,Y -28.613,Z -25.607,A 0.015,B 0.000,C 180.000} C_DIS
LIN {X -389.085,Y -27.648,Z -25.851,A 0.015,B -0.000,C 180.000} C_DIS
LIN {X -387.352,Y -21.275,Z -26.095,A 0.015,B 0.000,C 180.000} C_DIS
LIN {X -392.496,Y -17.133,Z -26.339,A 0.015,B 0.000,C 180.000} C_DIS
LIN {X -398.352,Y -20.187,Z -26.583,A 0.015,B -0.000,C -180.000} C_DIS
LIN {X -397.901,Y -26.776,Z -26.827,A 0.015,B -0.000,C -180.000} C_DIS
LIN {X -391.684,Y -29.003,Z -27.071,A 0.015,B -0.000,C 180.000} C_DIS
LIN {X -387.152,Y -24.199,Z -27.315,A 0.015,B -0.000,C -180.000} C_DIS
LIN {X -389.737,Y -18.122,Z -27.560,A 0.015,B 0.000,C -180.000} C_DIS
LIN {X -396.341,Y -18.055,Z -27.804,A 0.015,B 0.000,C 180.000} C_DIS
LIN {X -399.049,Y -24.079,Z -28.048,A 0.015,B 0.000,C 180.000} C_DIS
LIN {X -394.614,Y -28.973,Z -28.292,A 0.015,B -0.000,C -180.000} C_DIS
LIN {X -388.353,Y -26.872,Z -28.536,A 0.015,B 0.000,C 180.000} C_DIS
LIN {X -387.770,Y -20.293,Z -28.780,A 0.015,B 0.000,C -180.000} C_DIS
LIN {X -393.563,Y -17.122,Z -29.024,A 0.015,B 0.000,C -180.000} C_DIS
LIN {X -398.790,Y -21.160,Z -29.268,A 0.015,B -0.000,C -180.000} C_DIS
LIN {X -397.185,Y -27.566,Z -29.512,A 0.015,B 0.000,C 180.000} C_DIS
LIN {X -390.673,Y -28.663,Z -29.756,A 0.015,B -0.000,C 180.000} C_DIS
LIN {X -387.058,Y -23.136,Z -30.000,A 0.015,B 0.000,C -180.000} C_DIS
CIRC {X -392.664,Y -17.530,Z -30.000,A 0.015,B -0.000,C 180.000},{X -398.270,Y -23.137,Z -30.000,A 0.015,B -0.000,C -180.000} C_DIS
LIN {X -398.270,Y -23.645,Z -30.000,A 0.015,B 0.000,C -180.000} C_DIS
CIRC {X -397.651,Y -25.140,Z -30.000,A 0.015,B -0.000,C -180.000},{X -396.156,Y -25.759,Z -30.000,A 0.015,B 0.000,C 180.000} C_DIS
LIN {X -394.269,Y -25.759,Z -30.000,A 0.015,B 0.000,C -180.000} C_DIS
CIRC {X -392.505,Y -24.651,Z -30.000,A 0.015,B -0.000,C -180.000},{X -392.737,Y -22.582,Z -30.000,A 0.015,B 0.000,C -180.000} C_DIS
LIN {X -395.329,Y -19.326,Z -30.000,A 0.015,B -0.000,C -180.000} C_DIS
CIRC {X -397.164,Y -18.797,Z -30.000,A 0.015,B -0.000,C 180.000},{X -398.270,Y -20.354,Z -30.000,A 0.015,B -0.000,C -180.000} C_DIS
LIN {X -398.270,Y -23.137,Z -30.000,A 0.015,B 0.000,C -180.000} C_DIS
LIN {X -398.418,Y -23.660,Z -30.000,A 0.015,B -0.000,C 180.000} C_DIS
LIN {X -401.465,Y -28.615,Z -30.000,A 0.015,B 0.000,C 180.000} C_DIS
CIRC {X -402.315,Y -29.091,Z -30.000,A 0.015,B 0.000,C -180.000},{X -403.166,Y -28.618,Z -30.000,A 0.015,B 0.000,C 180.000} C_DIS
LIN {X -403.274,Y -28.444,Z -30.000,A 0.015,B 0.000,C -180.000} C_DIS
LIN {X -403.584,Y -27.623,Z -30.000,A 0.015,B 0.000,C 180.000} C_DIS
LIN {X -403.777,Y -26.414,Z -30.000,A 0.015,B -0.000,C 180.000} C_DIS
LIN {X -403.778,Y 7.523,Z -30.000,A 0.015,B 0.000,C -180.000} C_DIS
LIN {X -399.884,Y -2.513,Z -30.000,A 0.015,B -0.000,C 180.000} C_DIS
LIN {X -399.667,Y -2.969,Z -30.000,A 0.015,B 0.000,C -180.000} C_DIS
LIN {X -395.598,Y -10.084,Z -30.000,A 0.015,B 0.000,C -180.000} C_DIS
LIN {X -395.308,Y -10.512,Z -30.000,A 0.015,B 0.000,C -180.000} C_DIS
LIN {X -387.562,Y -20.241,Z -30.000,A 0.015,B -0.000,C -180.000} C_DIS
LIN {X -387.285,Y -20.548,Z -30.000,A 0.015,B 0.000,C -180.000} C_DIS
LIN {X -386.564,Y -21.256,Z -30.000,A 0.015,B 0.000,C -180.000} C_DIS
LIN {X -386.086,Y -21.646,Z -30.000,A 0.015,B 0.000,C -180.000} C_DIS
LIN {X -377.139,Y -27.680,Z -30.000,A 0.015,B 0.000,C 180.000} C_DIS
LIN {X -377.012,Y -27.761,Z -30.000,A 0.015,B -0.000,C 180.000} C_DIS
LIN {X -375.246,Y -28.842,Z -30.000,A 0.015,B -0.000,C 180.000} C_DIS
LIN {X -374.652,Y -29.130,Z -30.000,A 0.015,B 0.000,C -180.000} C_DIS
LIN {X -373.516,Y -29.549,Z -30.000,A 0.015,B 0.000,C -180.000} C_DIS
LIN {X -373.296,Y -29.621,Z -30.000,A 0.015,B -0.000,C -180.000} C_DIS
LIN {X -367.681,Y -31.266,Z -30.000,A 0.015,B 0.000,C 180.000} C_DIS
LIN {X -398.962,Y -31.266,Z -30.000,A 0.015,B -0.000,C 180.000} C_DIS
LIN {X -399.885,Y -31.140,Z -30.000,A 0.015,B 0.000,C 180.000} C_DIS
LIN {X -400.741,Y -30.861,Z -30.000,A 0.015,B 0.000,C 180.000} C_DIS
LIN {X -401.186,Y -30.616,Z -30.000,A 0.015,B 0.000,C -180.000} C_DIS
LIN {X -401.260,Y -29.552,Z -30.000,A 0.015,B -0.000,C 180.000} C_DIS
LIN {X -398.544,Y -27.508,Z -30.000,A 0.015,B -0.000,C -180.000} C_DIS
LIN {X -393.936,Y -23.884,Z -30.000,A 0.015,B 0.000,C 180.000} C_DIS
LIN {X -392.184,Y -23.292,Z -30.000,A 0.015,B -0.000,C -180.000} C_DIS
LIN {X -391.939,Y -22.804,Z -30.000,A 0.015,B 0.000,C 180.000} C_DIS
LIN {X -397.127,Y -18.723,Z -30.244,A 0.015,B -0.000,C 180.000} C_DIS
LIN {X -402.947,Y -21.837,Z -30.488,A 0.015,B -0.000,C 180.000} C_DIS
LIN {X -402.431,Y -28.417,Z -30.732,A 0.015,B 0.000,C 180.000} C_DIS
LIN {X -396.196,Y -30.585,Z -30.976,A 0.015,B 0.000,C 180.000} C_DIS
LIN {X -391.708,Y -25.745,Z -31.220,A 0.015,B -0.000,C -180.000} C_DIS
LIN {X -394.340,Y -19.692,Z -31.463,A 0.015,B -0.000,C -180.000} C_DIS
LIN {X -400.940,Y -19.673,Z -31.707,A 0.015,B -0.000,C -180.000} C_DIS
LIN {X -403.607,Y -25.711,Z -31.951,A 0.015,B 0.000,C 180.000} C_DIS
LIN {X -399.147,Y -30.577,Z -32.195,A 0.015,B -0.000,C -180.000} C_DIS
LIN {X -392.900,Y -28.445,Z -32.439,A 0.015,B -0.000,C -180.000} C_DIS
LIN {X -392.346,Y -21.867,Z -32.683,A 0.015,B 0.000,C 180.000} C_DIS
LIN {X -398.148,Y -18.720,Z -32.927,A 0.015,B -0.000,C -180.000} C_DIS
LIN {X -403.359,Y -22.771,Z -33.171,A 0.015,B 0.000,C -180.000} C_DIS
LIN {X -401.741,Y -29.170,Z -33.415,A 0.015,B -0.000,C 180.000} C_DIS
LIN {X -395.230,Y -30.256,Z -33.659,A 0.015,B 0.000,C -180.000} C_DIS
LIN {X -391.622,Y -24.728,Z -33.902,A 0.015,B 0.000,C 180.000} C_DIS
LIN {X -395.237,Y -19.205,Z -34.146,A 0.015,B -0.000,C 180.000} C_DIS
LIN {X -401.747,Y -20.300,Z -34.390,A 0.015,B 0.000,C 180.000} C_DIS
LIN {X -403.357,Y -26.701,Z -34.634,A 0.015,B -0.000,C -180.000} C_DIS
LIN {X -398.140,Y -30.745,Z -34.878,A 0.015,B -0.000,C -180.000} C_DIS
LIN {X -392.342,Y -27.590,Z -35.122,A 0.015,B 0.000,C -180.000} C_DIS
LIN {X -392.905,Y -21.013,Z -35.366,A 0.015,B 0.000,C -180.000} C_DIS
LIN {X -399.155,Y -18.889,Z -35.610,A 0.015,B 0.000,C -180.000} C_DIS
LIN {X -403.608,Y -23.761,Z -35.854,A 0.015,B -0.000,C -180.000} C_DIS
LIN {X -400.934,Y -29.796,Z -36.098,A 0.015,B 0.000,C -180.000} C_DIS
LIN {X -394.333,Y -29.768,Z -36.341,A 0.015,B -0.000,C -180.000} C_DIS
LIN {X -391.709,Y -23.710,Z -36.585,A 0.015,B 0.000,C -180.000} C_DIS
LIN {X -396.204,Y -18.876,Z -36.829,A 0.015,B -0.000,C -180.000} C_DIS
LIN {X -402.436,Y -21.053,Z -37.073,A 0.015,B -0.000,C 180.000} C_DIS
LIN {X -402.943,Y -27.635,Z -37.317,A 0.015,B -0.000,C -180.000} C_DIS
LIN {X -397.118,Y -30.741,Z -37.561,A 0.015,B 0.000,C -180.000} C_DIS
LIN {X -391.936,Y -26.653,Z -37.805,A 0.015,B 0.000,C 180.000} C_DIS
LIN {X -393.600,Y -20.265,Z -38.049,A 0.015,B 0.000,C -180.000} C_DIS
LIN {X -400.119,Y -19.226,Z -38.293,A 0.015,B 0.000,C 180.000} C_DIS
LIN {X -403.687,Y -24.779,Z -38.537,A 0.015,B 0.000,C -180.000} C_DIS
LIN {X -400.033,Y -30.276,Z -38.780,A 0.015,B 0.000,C 180.000} C_DIS
LIN {X -393.531,Y -29.135,Z -39.024,A 0.015,B 0.000,C -180.000} C_DIS
LIN {X -391.967,Y -22.722,Z -39.268,A 0.015,B -0.000,C -180.000} C_DIS
LIN {X -397.212,Y -18.716,Z -39.512,A 0.015,B -0.000,C -180.000} C_DIS
LIN {X -402.988,Y -21.912,Z -39.756,A 0.015,B 0.000,C 180.000} C_DIS
LIN {X -402.378,Y -28.485,Z -40.000,A 0.015,B 0.000,C 180.000} C_DIS
CIRC {X -394.501,Y -29.386,Z -40.000,A 0.015,B -0.000,C 180.000},{X -393.599,Y -21.510,Z -40.000,A 0.015,B 0.000,C 180.000} C_DIS
LIN {X -395.333,Y -19.328,Z -40.000,A 0.015,B 0.000,C 180.000} C_DIS
CIRC {X -397.167,Y -18.797,Z -40.000,A 0.015,B -0.000,C -180.000},{X -398.273,Y -20.354,Z -40.000,A 0.015,B -0.000,C 180.000} C_DIS
LIN {X -398.273,Y -23.648,Z -40.000,A 0.015,B 0.000,C -180.000} C_DIS
CIRC {X -397.653,Y -25.142,Z -40.000,A 0.015,B 0.000,C 180.000},{X -396.159,Y -25.761,Z -40.000,A 0.015,B 0.000,C 180.000} C_DIS
LIN {X -394.279,Y -25.761,Z -40.000,A 0.015,B 0.000,C -180.000} C_DIS
CIRC {X -392.515,Y -24.654,Z -40.000,A 0.015,B 0.000,C -180.000},{X -392.745,Y -22.584,Z -40.000,A 0.015,B 0.000,C 180.000} C_DIS
LIN {X -393.599,Y -21.510,Z -40.000,A 0.015,B 0.000,C 180.000} C_DIS
LIN {X -394.100,Y -21.130,Z -39.830,A 0.015,B 0.000,C -180.000} C_DIS
LIN {X -394.551,Y -21.030,Z -39.365,A 0.015,B 0.000,C 180.000} C_DIS
LIN {X -394.721,Y -21.036,Z -38.730,A 0.015,B -0.000,C 180.000} C_DIS
$VEL.CP = 1.00000
LIN {X -394.721,Y -21.036,Z 11.000,A 0.015,B -0.000,C 180.000} C_DIS
$VEL.CP = 1.00000
LIN {X -396.980,Y -23.891,Z 11.000,A 0.015,B 0.000,C -180.000} C_DIS
$VEL.CP = 0.10000
LIN {X -396.980,Y -23.891,Z -19.000,A 0.015,B 0.000,C -180.000} C_DIS
LIN {X -396.980,Y -23.891,Z -38.730,A 0.015,B -0.000,C 180.000} C_DIS
LIN {X -398.086,Y -24.516,Z -40.000,A 0.015,B -0.000,C -180.000} C_DIS
LIN {X -403.584,Y -27.623,Z -40.000,A 0.015,B 0.000,C -180.000} C_DIS
LIN {X -403.777,Y -26.414,Z -40.000,A 0.015,B 0.000,C -180.000} C_DIS
LIN {X -403.778,Y 7.523,Z -40.000,A 0.015,B 0.000,C -180.000} C_DIS
LIN {X -399.884,Y -2.513,Z -40.000,A 0.015,B -0.000,C 180.000} C_DIS
LIN {X -399.667,Y -2.969,Z -40.000,A 0.015,B -0.000,C -180.000} C_DIS
LIN {X -395.598,Y -10.084,Z -40.000,A 0.015,B 0.000,C -180.000} C_DIS
LIN {X -395.310,Y -10.510,Z -40.000,A 0.015,B 0.000,C 180.000} C_DIS
LIN {X -387.579,Y -20.238,Z -40.000,A 0.015,B 0.000,C -180.000} C_DIS
LIN {X -387.276,Y -20.571,Z -40.000,A 0.015,B 0.000,C -180.000} C_DIS
LIN {X -386.544,Y -21.276,Z -40.000,A 0.015,B -0.000,C 180.000} C_DIS
LIN {X -386.093,Y -21.640,Z -40.000,A 0.015,B 0.000,C 180.000} C_DIS
LIN {X -376.259,Y -28.291,Z -40.000,A 0.015,B 0.000,C -180.000} C_DIS
LIN {X -375.911,Y -28.498,Z -40.000,A 0.015,B 0.000,C 180.000} C_DIS
LIN {X -374.744,Y -29.098,Z -40.000,A 0.015,B 0.000,C 180.000} C_DIS
LIN {X -374.209,Y -29.317,Z -40.000,A 0.015,B 0.000,C -180.000} C_DIS
LIN {X -370.455,Y -30.494,Z -40.000,A 0.015,B -0.000,C 180.000} C_DIS
LIN {X -370.397,Y -30.512,Z -40.000,A 0.015,B -0.000,C -180.000} C_DIS
LIN {X -367.833,Y -31.266,Z -40.000,A 0.015,B 0.000,C 180.000} C_DIS
LIN {X -398.962,Y -31.266,Z -40.000,A 0.015,B -0.000,C 180.000} C_DIS
LIN {X -399.885,Y -31.140,Z -40.000,A 0.015,B 0.000,C 180.000} C_DIS
LIN {X -400.741,Y -30.861,Z -40.000,A 0.015,B -0.000,C -180.000} C_DIS
LIN {X -401.186,Y -30.616,Z -40.000,A 0.015,B 0.000,C 180.000} C_DIS
LIN {X -401.088,Y -28.818,Z -40.000,A 0.015,B 0.000,C -180.000} C_DIS
LIN {X -392.101,Y -25.032,Z -40.000,A 0.015,B 0.000,C 180.000} C_DIS
LIN {X -389.721,Y -19.058,Z -40.237,A 0.015,B -0.000,C 180.000} C_DIS
LIN {X -394.083,Y -14.332,Z -40.474,A 0.015,B 0.000,C 180.000} C_DIS
LIN {X -400.228,Y -16.225,Z -40.711,A 0.015,B -0.000,C -180.000} C_DIS
LIN {X -401.175,Y -22.586,Z -40.947,A 0.015,B 0.000,C -180.000} C_DIS
LIN {X -395.846,Y -26.186,Z -41.184,A 0.015,B -0.000,C 180.000} C_DIS
LIN {X -390.298,Y -22.934,Z -41.421,A 0.015,B -0.000,C 180.000} C_DIS
LIN {X -390.835,Y -16.526,Z -41.658,A 0.015,B 0.000,C 180.000} C_DIS
LIN {X -396.847,Y -14.243,Z -41.895,A 0.015,B 0.000,C -180.000} C_DIS
LIN {X -401.502,Y -18.680,Z -42.132,A 0.015,B 0.000,C 180.000} C_DIS
LIN {X -399.511,Y -24.794,Z -42.368,A 0.015,B 0.000,C -180.000} C_DIS
LIN {X -393.136,Y -25.639,Z -42.605,A 0.015,B -0.000,C 180.000} C_DIS
LIN {X -389.621,Y -20.253,Z -42.842,A 0.015,B -0.000,C -180.000} C_DIS
LIN {X -392.961,Y -14.758,Z -43.079,A 0.015,B 0.000,C -180.000} C_DIS
LIN {X -399.360,Y -15.397,Z -43.316,A 0.015,B -0.000,C 180.000} C_DIS
LIN {X -401.546,Y -21.445,Z -43.553,A 0.015,B 0.000,C -180.000} C_DIS
LIN {X -397.036,Y -26.028,Z -43.789,A 0.015,B -0.000,C 180.000} C_DIS
LIN {X -390.954,Y -23.939,Z -44.026,A 0.015,B 0.000,C -180.000} C_DIS
LIN {X -390.212,Y -17.551,Z -44.263,A 0.015,B 0.000,C 180.000} C_DIS
LIN {X -395.653,Y -14.124,Z -44.500,A 0.015,B 0.000,C -180.000} C_DIS
CIRC {X -401.472,Y -19.943,Z -44.500,A 0.015,B 0.000,C 180.000},{X -395.653,Y -25.762,Z -44.500,A 0.015,B 0.000,C -180.000} C_DIS
LIN {X -394.283,Y -25.762,Z -44.500,A 0.015,B -0.000,C -180.000} C_DIS
CIRC {X -392.519,Y -24.655,Z -44.500,A 0.015,B 0.000,C 180.000},{X -392.749,Y -22.585,Z -44.500,A 0.015,B -0.000,C -180.000} C_DIS
LIN {X -395.334,Y -19.329,Z -44.500,A 0.015,B 0.000,C 180.000} C_DIS
CIRC {X -397.168,Y -18.798,Z -44.500,A 0.015,B 0.000,C 180.000},{X -398.274,Y -20.354,Z -44.500,A 0.015,B -0.000,C 180.000} C_DIS
LIN {X -398.274,Y -23.649,Z -44.500,A 0.015,B 0.000,C 180.000} C_DIS
CIRC {X -397.654,Y -25.143,Z -44.500,A 0.015,B 0.000,C 180.000},{X -396.160,Y -25.762,Z -44.500,A 0.015,B 0.000,C 180.000} C_DIS
LIN {X -395.653,Y -25.762,Z -44.500,A 0.015,B 0.000,C 180.000} C_DIS
LIN {X -395.469,Y -27.745,Z -44.500,A 0.015,B 0.000,C 180.000} C_DIS
LIN {X -400.886,Y -28.757,Z -44.500,A 0.015,B 0.000,C -180.000} C_DIS
LIN {X -401.186,Y -30.616,Z -44.500,A 0.015,B -0.000,C -180.000} C_DIS
LIN {X -400.741,Y -30.861,Z -44.500,A 0.015,B 0.000,C -180.000} C_DIS
LIN {X -399.885,Y -31.140,Z -44.500,A 0.015,B 0.000,C -180.000} C_DIS
LIN {X -398.962,Y -31.266,Z -44.500,A 0.015,B 0.000,C -180.000} C_DIS
LIN {X -367.794,Y -31.266,Z -44.500,A 0.015,B 0.000,C 180.000} C_DIS
LIN {X -373.885,Y -29.439,Z -44.500,A 0.015,B 0.000,C 180.000} C_DIS
LIN {X -374.378,Y -29.248,Z -44.500,A 0.015,B 0.000,C -180.000} C_DIS
LIN {X -375.830,Y -28.550,Z -44.500,A 0.015,B 0.000,C 180.000} C_DIS
LIN {X -376.262,Y -28.302,Z -44.500,A 0.015,B -0.000,C -180.000} C_DIS
LIN {X -386.097,Y -21.637,Z -44.500,A 0.015,B 0.000,C 180.000} C_DIS
LIN {X -386.536,Y -21.284,Z -44.500,A 0.015,B 0.000,C 180.000} C_DIS
LIN {X -387.272,Y -20.581,Z -44.500,A 0.015,B -0.000,C 180.000} C_DIS
LIN {X -387.586,Y -20.237,Z -44.500,A 0.015,B -0.000,C 180.000} C_DIS
LIN {X -395.310,Y -10.509,Z -44.500,A 0.015,B -0.000,C 180.000} C_DIS
LIN {X -395.598,Y -10.084,Z -44.500,A 0.015,B 0.000,C 180.000} C_DIS
LIN {X -399.667,Y -2.969,Z -44.500,A 0.015,B -0.000,C -180.000} C_DIS
LIN {X -399.881,Y -2.522,Z -44.500,A 0.015,B 0.000,C 180.000} C_DIS
LIN {X -403.778,Y 7.441,Z -44.500,A 0.015,B -0.000,C -180.000} C_DIS
LIN {X -403.777,Y -26.414,Z -44.500,A 0.015,B 0.000,C 180.000} C_DIS
LIN {X -403.584,Y -27.623,Z -44.500,A 0.015,B 0.000,C -180.000} C_DIS
LIN {X -403.274,Y -28.444,Z -44.500,A 0.015,B -0.000,C 180.000} C_DIS
LIN {X -403.166,Y -28.618,Z -44.500,A 0.015,B 0.000,C -180.000} C_DIS
LIN {X -402.571,Y -28.706,Z -44.500,A 0.015,B 0.000,C 180.000} C_DIS
LIN {X -401.121,Y -27.438,Z -44.500,A 0.015,B 0.000,C 180.000} C_DIS
LIN {X -394.754,Y -24.028,Z -44.500,A 0.015,B 0.000,C -180.000} C_DIS
LIN {X -392.320,Y -23.476,Z -44.500,A 0.015,B -0.000,C 180.000} C_DIS
LIN {X -391.944,Y -22.813,Z -44.500,A 0.015,B -0.000,C -180.000} C_DIS
LIN {X -397.127,Y -18.726,Z -44.744,A 0.015,B 0.000,C 180.000} C_DIS
LIN {X -402.951,Y -21.834,Z -44.988,A 0.015,B 0.000,C 180.000} C_DIS
LIN {X -402.442,Y -28.415,Z -45.232,A 0.015,B -0.000,C -180.000} C_DIS
LIN {X -396.210,Y -30.590,Z -45.476,A 0.015,B 0.000,C -180.000} C_DIS
LIN {X -391.716,Y -25.755,Z -45.720,A 0.015,B 0.000,C 180.000} C_DIS
LIN {X -394.341,Y -19.699,Z -45.963,A 0.015,B -0.000,C -180.000} C_DIS
LIN {X -400.942,Y -19.672,Z -46.207,A 0.015,B 0.000,C 180.000} C_DIS
LIN {X -403.615,Y -25.707,Z -46.451,A 0.015,B -0.000,C -180.000} C_DIS
LIN {X -399.161,Y -30.578,Z -46.695,A 0.015,B 0.000,C -180.000} C_DIS
LIN {X -392.911,Y -28.453,Z -46.939,A 0.015,B 0.000,C 180.000} C_DIS
LIN {X -392.350,Y -21.876,Z -47.183,A 0.015,B 0.000,C 180.000} C_DIS
LIN {X -398.148,Y -18.722,Z -47.427,A 0.015,B 0.000,C 180.000} C_DIS
LIN {X -403.364,Y -22.767,Z -47.671,A 0.015,B -0.000,C 180.000} C_DIS
LIN {X -401.753,Y -29.168,Z -47.915,A 0.015,B 0.000,C 180.000} C_DIS
LIN {X -395.243,Y -30.261,Z -48.159,A 0.015,B 0.000,C -180.000} C_DIS
LIN {X -391.629,Y -24.738,Z -48.402,A 0.015,B 0.000,C -180.000} C_DIS
LIN {X -395.238,Y -19.211,Z -48.646,A 0.015,B 0.000,C -180.000} C_DIS
LIN {X -401.749,Y -20.298,Z -48.890,A 0.015,B 0.000,C 180.000} C_DIS
LIN {X -403.366,Y -26.698,Z -49.134,A 0.015,B 0.000,C 180.000} C_DIS
LIN {X -398.154,Y -30.747,Z -49.378,A 0.015,B 0.000,C 180.000} C_DIS
LIN {X -392.352,Y -27.599,Z -49.622,A 0.015,B 0.000,C 180.000} C_DIS
LIN {X -392.908,Y -21.021,Z -49.866,A 0.015,B 0.000,C 180.000} C_DIS
LIN {X -399.155,Y -18.890,Z -50.110,A 0.015,B 0.000,C 180.000} C_DIS
LIN {X -403.615,Y -23.757,Z -50.354,A 0.015,B 0.000,C -180.000} C_DIS
LIN {X -400.946,Y -29.795,Z -50.598,A 0.015,B 0.000,C 180.000} C_DIS
LIN {X -394.346,Y -29.774,Z -50.841,A 0.015,B -0.000,C 180.000} C_DIS
LIN {X -391.715,Y -23.720,Z -51.085,A 0.015,B 0.000,C -180.000} C_DIS
LIN {X -396.205,Y -18.881,Z -51.329,A 0.015,B -0.000,C 180.000} C_DIS
LIN {X -402.439,Y -21.051,Z -51.573,A 0.015,B 0.000,C -180.000} C_DIS
LIN {X -402.953,Y -27.632,Z -51.817,A 0.015,B -0.000,C 180.000} C_DIS
LIN {X -397.133,Y -30.744,Z -52.061,A 0.015,B 0.000,C -180.000} C_DIS
LIN {X -391.945,Y -26.662,Z -52.305,A 0.015,B 0.000,C 180.000} C_DIS
LIN {X -393.603,Y -20.273,Z -52.549,A 0.015,B -0.000,C 180.000} C_DIS
LIN {X -400.120,Y -19.226,Z -52.793,A 0.015,B 0.000,C 180.000} C_DIS
LIN {X -403.694,Y -24.775,Z -53.037,A 0.015,B 0.000,C -180.000} C_DIS
LIN {X -400.046,Y -30.276,Z -53.280,A 0.015,B 0.000,C 180.000} C_DIS
LIN {X -393.543,Y -29.143,Z -53.524,A 0.015,B 0.000,C -180.000} C_DIS
LIN {X -391.972,Y -22.732,Z -53.768,A 0.015,B 0.000,C 180.000} C_DIS
LIN {X -397.213,Y -18.719,Z -54.012,A 0.015,B 0.000,C 180.000} C_DIS
LIN {X -402.992,Y -21.909,Z -54.256,A 0.015,B 0.000,C -180.000} C_DIS
LIN {X -402.389,Y -28.483,Z -54.500,A 0.015,B 0.000,C 180.000} C_DIS
CIRC {X -398.640,Y -30.569,Z -54.500,A 0.015,B 0.000,C -180.000},{X -394.514,Y -29.393,Z -54.500,A 0.015,B 0.000,C -180.000} C_DIS
CIRC {X -392.427,Y -25.644,Z -54.500,A 0.015,B -0.000,C 180.000},{X -393.603,Y -21.517,Z -54.500,A 0.015,B 0.000,C 180.000} C_DIS
LIN {X -395.337,Y -19.330,Z -54.500,A 0.015,B 0.000,C -180.000} C_DIS
CIRC {X -397.170,Y -18.798,Z -54.500,A 0.015,B 0.000,C -180.000},{X -398.276,Y -20.354,Z -54.500,A 0.015,B -0.000,C -180.000} C_DIS
LIN {X -398.276,Y -23.651,Z -54.500,A 0.015,B 0.000,C 180.000} C_DIS
CIRC {X -397.656,Y -25.145,Z -54.500,A 0.015,B 0.000,C -180.000},{X -396.162,Y -25.764,Z -54.500,A 0.015,B 0.000,C 180.000} C_DIS
LIN {X -394.291,Y -25.764,Z -54.500,A 0.015,B 0.000,C -180.000} C_DIS
CIRC {X -392.526,Y -24.658,Z -54.500,A 0.015,B 0.000,C -180.000},{X -392.755,Y -22.587,Z -54.500,A 0.015,B 0.000,C -180.000} C_DIS
LIN {X -393.603,Y -21.517,Z -54.500,A 0.015,B 0.000,C -180.000} C_DIS
LIN {X -394.103,Y -21.137,Z -54.330,A 0.015,B 0.000,C 180.000} C_DIS
LIN {X -394.555,Y -21.037,Z -53.865,A 0.015,B -0.000,C -180.000} C_DIS
LIN {X -394.725,Y -21.043,Z -53.230,A 0.015,B 0.000,C -180.000} C_DIS
$VEL.CP = 1.00000
LIN {X -394.725,Y -21.043,Z 11.000,A 0.015,B -0.000,C -180.000} C_DIS
$VEL.CP = 1.00000
LIN {X -396.503,Y -24.430,Z 11.000,A 0.015,B -0.000,C 180.000} C_DIS
$VEL.CP = 0.10000
LIN {X -396.503,Y -24.430,Z -33.500,A 0.015,B -0.000,C -180.000} C_DIS
LIN {X -396.503,Y -24.430,Z -53.230,A 0.015,B -0.000,C -180.000} C_DIS
LIN {X -397.202,Y -25.491,Z -54.500,A 0.015,B 0.000,C 180.000} C_DIS
LIN {X -400.741,Y -30.861,Z -54.500,A 0.015,B 0.000,C 180.000} C_DIS
LIN {X -399.885,Y -31.140,Z -54.500,A 0.015,B 0.000,C -180.000} C_DIS
LIN {X -398.962,Y -31.266,Z -54.500,A 0.015,B 0.000,C -180.000} C_DIS
LIN {X -367.821,Y -31.266,Z -54.500,A 0.015,B 0.000,C 180.000} C_DIS
LIN {X -374.184,Y -29.325,Z -54.500,A 0.015,B -0.000,C 180.000} C_DIS
LIN {X -374.676,Y -29.132,Z -54.500,A 0.015,B 0.000,C 180.000} C_DIS
LIN {X -375.843,Y -28.565,Z -54.500,A 0.015,B -0.000,C -180.000} C_DIS
LIN {X -376.266,Y -28.320,Z -54.500,A 0.015,B 0.000,C -180.000} C_DIS
LIN {X -386.104,Y -21.632,Z -54.500,A 0.015,B -0.000,C -180.000} C_DIS
LIN {X -386.520,Y -21.299,Z -54.500,A 0.015,B 0.000,C 180.000} C_DIS
LIN {X -387.265,Y -20.599,Z -54.500,A 0.015,B -0.000,C 180.000} C_DIS
LIN {X -387.599,Y -20.235,Z -54.500,A 0.015,B 0.000,C -180.000} C_DIS
LIN {X -395.312,Y -10.507,Z -54.500,A 0.015,B 0.000,C -180.000} C_DIS
LIN {X -395.598,Y -10.084,Z -54.500,A 0.015,B -0.000,C 180.000} C_DIS
LIN {X -399.667,Y -2.969,Z -54.500,A 0.015,B 0.000,C 180.000} C_DIS
LIN {X -399.881,Y -2.522,Z -54.500,A 0.015,B 0.000,C 180.000} C_DIS
LIN {X -403.778,Y 7.434,Z -54.500,A 0.015,B -0.000,C 180.000} C_DIS
LIN {X -403.777,Y -26.414,Z -54.500,A 0.015,B 0.000,C 180.000} C_DIS
LIN {X -403.584,Y -27.623,Z -54.500,A 0.015,B 0.000,C 180.000} C_DIS
LIN {X -403.274,Y -28.444,Z -54.500,A 0.015,B -0.000,C 180.000} C_DIS
LIN {X -403.166,Y -28.618,Z -54.500,A 0.015,B 0.000,C -180.000} C_DIS
LIN {X -402.571,Y -28.706,Z -54.500,A 0.015,B 0.000,C -180.000} C_DIS
LIN {X -401.121,Y -27.438,Z -54.500,A 0.015,B 0.000,C 180.000} C_DIS
LIN {X -394.757,Y -24.031,Z -54.500,A 0.015,B 0.000,C -180.000} C_DIS
LIN {X -392.323,Y -23.481,Z -54.500,A 0.015,B -0.000,C 180.000} C_DIS
LIN {X -391.946,Y -22.818,Z -54.500,A 0.015,B 0.000,C -180.000} C_DIS
LIN {X -397.127,Y -18.728,Z -54.744,A 0.015,B 0.000,C 180.000} C_DIS
LIN {X -402.953,Y -21.832,Z -54.988,A 0.015,B 0.000,C 180.000} C_DIS
LIN {X -402.448,Y -28.414,Z -55.232,A 0.015,B -0.000,C 180.000} C_DIS
LIN {X -396.217,Y -30.593,Z -55.476,A 0.015,B 0.000,C -180.000} C_DIS
LIN {X -391.721,Y -25.760,Z -55.720,A 0.015,B 0.000,C 180.000} C_DIS
LIN {X -394.342,Y -19.702,Z -55.963,A 0.015,B 0.000,C -180.000} C_DIS
LIN {X -400.943,Y -19.672,Z -56.207,A 0.015,B 0.000,C -180.000} C_DIS
LIN {X -403.620,Y -25.705,Z -56.451,A 0.015,B 0.000,C -180.000} C_DIS
LIN {X -399.168,Y -30.579,Z -56.695,A 0.015,B -0.000,C -180.000} C_DIS
LIN {X -392.918,Y -28.458,Z -56.939,A 0.015,B 0.000,C 180.000} C_DIS
LIN {X -392.352,Y -21.881,Z -57.183,A 0.015,B 0.000,C 180.000} C_DIS
LIN {X -398.149,Y -18.723,Z -57.427,A 0.015,B 0.000,C -180.000} C_DIS
LIN {X -403.367,Y -22.765,Z -57.671,A 0.015,B 0.000,C 180.000} C_DIS
LIN {X -401.759,Y -29.167,Z -57.915,A 0.015,B -0.000,C 180.000} C_DIS
LIN {X -395.250,Y -30.264,Z -58.159,A 0.015,B 0.000,C 180.000} C_DIS
LIN {X -391.633,Y -24.743,Z -58.402,A 0.015,B 0.000,C -180.000} C_DIS
LIN {X -395.239,Y -19.214,Z -58.646,A 0.015,B 0.000,C 180.000} C_DIS
LIN {X -401.750,Y -20.297,Z -58.890,A 0.015,B 0.000,C 180.000} C_DIS
LIN {X -403.371,Y -26.696,Z -59.134,A 0.015,B 0.000,C -180.000} C_DIS
LIN {X -398.161,Y -30.749,Z -59.378,A 0.015,B 0.000,C 180.000} C_DIS
LIN {X -392.358,Y -27.603,Z -59.622,A 0.015,B -0.000,C 180.000} C_DIS
LIN {X -392.910,Y -21.026,Z -59.866,A 0.015,B 0.000,C 180.000} C_DIS
LIN {X -399.156,Y -18.891,Z -60.110,A 0.015,B -0.000,C 180.000} C_DIS
LIN {X -403.618,Y -23.755,Z -60.354,A 0.015,B 0.000,C 180.000} C_DIS
LIN {X -400.953,Y -29.794,Z -60.598,A 0.015,B 0.000,C -180.000} C_DIS
LIN {X -394.353,Y -29.778,Z -60.841,A 0.015,B 0.000,C 180.000} C_DIS
LIN {X -391.719,Y -23.725,Z -61.085,A 0.015,B 0.000,C -180.000} C_DIS
LIN {X -396.205,Y -18.884,Z -61.329,A 0.015,B 0.000,C -180.000} C_DIS
LIN {X -402.440,Y -21.050,Z -61.573,A 0.015,B -0.000,C 180.000} C_DIS
LIN {X -402.959,Y -27.630,Z -61.817,A 0.015,B 0.000,C -180.000} C_DIS
LIN {X -397.140,Y -30.746,Z -62.061,A 0.015,B 0.000,C -180.000} C_DIS
LIN {X -391.950,Y -26.667,Z -62.305,A 0.015,B 0.000,C 180.000} C_DIS
LIN {X -393.604,Y -20.277,Z -62.549,A 0.015,B -0.000,C 180.000} C_DIS
LIN {X -400.120,Y -19.226,Z -62.793,A 0.015,B 0.000,C 180.000} C_DIS
LIN {X -403.698,Y -24.773,Z -63.037,A 0.015,B 0.000,C 180.000} C_DIS
LIN {X -400.053,Y -30.277,Z -63.280,A 0.015,B -0.000,C 180.000} C_DIS
LIN {X -393.550,Y -29.147,Z -63.524,A 0.015,B 0.000,C 180.000} C_DIS
LIN {X -391.974,Y -22.737,Z -63.768,A 0.015,B 0.000,C 180.000} C_DIS
LIN {X -397.213,Y -18.721,Z -64.012,A 0.015,B 0.000,C 180.000} C_DIS
LIN {X -402.994,Y -21.908,Z -64.256,A 0.015,B -0.000,C -180.000} C_DIS
LIN {X -402.395,Y -28.481,Z -64.500,A 0.015,B -0.000,C 180.000} C_DIS
CIRC {X -394.520,Y -29.396,Z -64.500,A 0.015,B -0.000,C -180.000},{X -393.605,Y -21.522,Z -64.500,A 0.015,B 0.000,C -180.000} C_DIS
LIN {X -395.339,Y -19.332,Z -64.500,A 0.015,B 0.000,C -180.000} C_DIS
CIRC {X -397.172,Y -18.799,Z -64.500,A 0.015,B 0.000,C -180.000},{X -398.277,Y -20.354,Z -64.500,A 0.015,B 0.000,C -180.000} C_DIS
LIN {X -398.277,Y -23.652,Z -64.500,A 0.015,B 0.000,C 180.000} C_DIS
CIRC {X -397.658,Y -25.147,Z -64.500,A 0.015,B -0.000,C 180.000},{X -396.163,Y -25.766,Z -64.500,A 0.015,B -0.000,C 180.000} C_DIS
LIN {X -394.297,Y -25.766,Z -64.500,A 0.015,B 0.000,C -180.000} C_DIS
CIRC {X -392.532,Y -24.659,Z -64.500,A 0.015,B 0.000,C 180.000},{X -392.760,Y -22.589,Z -64.500,A 0.015,B -0.000,C -180.000} C_DIS
LIN {X -393.605,Y -21.522,Z -64.500,A 0.015,B -0.000,C 180.000} C_DIS
CIRC {X -394.378,Y -21.142,Z -64.500,A 0.015,B -0.000,C 180.000},{X -395.159,Y -21.503,Z -64.500,A 0.015,B 0.000,C -180.000} C_DIS
LIN {X -401.471,Y -29.101,Z -64.500,A 0.015,B 0.000,C -180.000} C_DIS
LIN {X -401.186,Y -30.616,Z -64.500,A 0.015,B -0.000,C -180.000} C_DIS
LIN {X -400.741,Y -30.861,Z -64.500,A 0.015,B 0.000,C -180.000} C_DIS
LIN {X -399.885,Y -31.140,Z -64.500,A 0.015,B -0.000,C -180.000} C_DIS
LIN {X -398.962,Y -31.266,Z -64.500,A 0.015,B 0.000,C 180.000} C_DIS
LIN {X -367.907,Y -31.266,Z -64.500,A 0.015,B 0.000,C 180.000} C_DIS
LIN {X -374.197,Y -29.321,Z -64.500,A 0.015,B 0.000,C -180.000} C_DIS
LIN {X -374.741,Y -29.099,Z -64.500,A 0.015,B 0.000,C 180.000} C_DIS
LIN {X -376.349,Y -28.275,Z -64.500,A 0.015,B 0.000,C -180.000} C_DIS
LIN {X -376.726,Y -28.049,Z -64.500,A 0.015,B 0.000,C 180.000} C_DIS
LIN {X -386.376,Y -21.396,Z -64.500,A 0.015,B -0.000,C -180.000} C_DIS
LIN {X -386.787,Y -21.062,Z -64.500,A 0.015,B 0.000,C 180.000} C_DIS
LIN {X -387.289,Y -20.585,Z -64.500,A 0.015,B 0.000,C -180.000} C_DIS
LIN {X -387.610,Y -20.234,Z -64.500,A 0.015,B 0.000,C 180.000} C_DIS
LIN {X -395.313,Y -10.505,Z -64.500,A 0.015,B 0.000,C 180.000} C_DIS
LIN {X -395.598,Y -10.084,Z -64.500,A 0.015,B 0.000,C 180.000} C_DIS
LIN {X -399.667,Y -2.969,Z -64.500,A 0.015,B 0.000,C -180.000} C_DIS
LIN {X -399.877,Y -2.530,Z -64.500,A 0.015,B 0.000,C 180.000} C_DIS
LIN {X -403.778,Y 7.361,Z -64.500,A 0.015,B 0.000,C -180.000} C_DIS
LIN {X -403.777,Y -26.414,Z -64.500,A 0.015,B -0.000,C -180.000} C_DIS
LIN {X -403.584,Y -27.623,Z -64.500,A 0.015,B 0.000,C 180.000} C_DIS
LIN {X -403.274,Y -28.444,Z -64.500,A 0.015,B 0.000,C 180.000} C_DIS
LIN {X -403.166,Y -28.618,Z -64.500,A 0.015,B 0.000,C 180.000} C_DIS
LIN {X -402.713,Y -29.054,Z -64.330,A 0.015,B 0.000,C 180.000} C_DIS
LIN {X -402.276,Y -29.205,Z -63.865,A 0.015,B 0.000,C 180.000} C_DIS
LIN {X -402.107,Y -29.218,Z -63.230,A 0.015,B 0.000,C -180.000} C_DIS
$VEL.CP = 1.00000
LIN {X -402.107,Y -29.218,Z 15.000,A 0.015,B 0.000,C -180.000} C_DIS
$VEL.CP = 1.00000
LIN {X -402.107,Y -29.218,Z 15.000,A 0.015,B 0.000,C -180.000} C_DIS
END
